(* IEC 61131-3 sources: AxTestProject/Program/AuxFunc, 3 files *)

(* ---- tDefaults.st ---- *)
TYPE
    tDefaults : Struct
        a : int := 1;
        b : INT := 2;
        c : BOOL := true;
    END_STRUCT;
END_TYPE

TYPE
    Motor : STRUCT
        setPointSpeed : LREAL := 30.0;
        error, speed, lastSpeed : LREAL;
    END_STRUCT;
END_TYPE

TYPE
    nArray : ARRAY[0..9] of INT := [1, 2, 3, 4, 5, 6, 7, 8, 9, 10];

END_TYPE

(* ---- add.st ---- *)
FUNCTION add2 : Int
    VAR_INPUT
        s1 : INT;
        s2 : INT;
    END_VAR
    VAR_TEMP
    END_VAR
        add2 := s1 + s2;
        ;
END_FUNCTION

(* ---- test.st ---- *)
NAMESPACE A
    NAMESPACE  Aa
        FUNCTION inner : Int
            VAR_INPUT
            END_VAR
            VAR_TEMP
            END_VAR
            inner := 1;
                            ;
        END_FUNCTION
    END_NAMESPACE
    FUNCTION test : Int
        VAR_INPUT
        END_VAR
        VAR_TEMP
        END_VAR
        B.test();
        test  := 0;
            ;
    END_FUNCTION
END_NAMESPACE

NAMESPACE B
    FUNCTION test : Int
        VAR_INPUT
        END_VAR
        VAR_TEMP
        END_VAR
           A.aa.inner();
            test := 1;
            ;
    END_FUNCTION

END_NAMESPACE
